// ---- POUs/MAIN.TcPOU
PROGRAM MAIN
VAR
	fbXTSSystem : XTS_System;
	bInit		: BOOL := FALSE;
	i : UDINT;
END_VAR

IF bInit = FALSE THEN
	
		fbXTSSystem.stCfg.bInvertPolarity						:= FALSE;
	
		fbXTSSystem.stCfg.udiNumStations						:= 7;
		fbXTSSystem.stCfg.stStationsCfg[1].sName			 	:= 'Station 1'; 
		fbXTSSystem.stCfg.stStationsCfg[1].lrStartPosition 		:= 0.0; 
		fbXTSSystem.stCfg.stStationsCfg[1].lrEndPosition	 	:= 500.0; 
		fbXTSSystem.stCfg.stStationsCfg[1].lrStopPosition[1] 	:= 100.0; 
		fbXTSSystem.stCfg.stStationsCfg[1].lrStopPosition[2] 	:= 350.0; 
		fbXTSSystem.stCfg.stStationsCfg[1].lrProcessingTime 	:= 2.0;
		fbXTSSystem.stCfg.stStationsCfg[1].uiNumStopPositions 	:= 2;
		fbXTSSystem.stCfg.stStationsCfg[1].lrTravelTime			:= 0.5;				

		fbXTSSystem.stCfg.stStationsCfg[2].sName			 	:= 'Station 2'; 		
		fbXTSSystem.stCfg.stStationsCfg[2].lrStartPosition 		:= 1000.0; 
		fbXTSSystem.stCfg.stStationsCfg[2].lrEndPosition	 	:= 1500.0;
		fbXTSSystem.stCfg.stStationsCfg[2].lrStopPosition[1]	:= 10.0; 
		fbXTSSystem.stCfg.stStationsCfg[2].lrStopPosition[2]	:= 400.0; 
		fbXTSSystem.stCfg.stStationsCfg[2].lrStopPosition[3]	:= 500.0; 
		fbXTSSystem.stCfg.stStationsCfg[2].lrProcessingTime 	:= 3.0;
		fbXTSSystem.stCfg.stStationsCfg[2].uiNumStopPositions 	:= 2;
		fbXTSSystem.stCfg.stStationsCfg[2].lrTravelTime			:= 0.5;				

 		fbXTSSystem.stCfg.stStationsCfg[3].sName			 	:= 'Station 3';  
		fbXTSSystem.stCfg.stStationsCfg[3].lrStartPosition 		:= 2000.0; 
		fbXTSSystem.stCfg.stStationsCfg[3].lrEndPosition	 	:= 2500.0;
		fbXTSSystem.stCfg.stStationsCfg[3].lrStopPosition[1] 	:= 100.0; 
		fbXTSSystem.stCfg.stStationsCfg[3].lrProcessingTime 	:= 1.0;
		fbXTSSystem.stCfg.stStationsCfg[3].uiNumStopPositions 	:= 1;
		fbXTSSystem.stCfg.stStationsCfg[3].lrTravelTime			:= 0.5;				

		fbXTSSystem.stCfg.stStationsCfg[4].sName			 	:= 'Station 4'; 	
		fbXTSSystem.stCfg.stStationsCfg[4].lrStartPosition 		:= 3000.0; 
		fbXTSSystem.stCfg.stStationsCfg[4].lrEndPosition	 	:= 3500.0;
		fbXTSSystem.stCfg.stStationsCfg[4].lrStopPosition[1] 	:= 200.0; 
		fbXTSSystem.stCfg.stStationsCfg[4].lrProcessingTime 	:= 1.0;
		fbXTSSystem.stCfg.stStationsCfg[4].uiNumStopPositions 	:= 1;
		fbXTSSystem.stCfg.stStationsCfg[4].lrTravelTime			:= 0.5;				

		fbXTSSystem.stCfg.stStationsCfg[5].sName			 	:= 'Station 5'; 
		fbXTSSystem.stCfg.stStationsCfg[5].lrStartPosition 		:= 4000.0; 
		fbXTSSystem.stCfg.stStationsCfg[5].lrEndPosition	 	:= 4500.0;
		fbXTSSystem.stCfg.stStationsCfg[5].lrStopPosition[1] 	:= 300.0; 
		fbXTSSystem.stCfg.stStationsCfg[5].lrProcessingTime 	:= 1.0;
		fbXTSSystem.stCfg.stStationsCfg[5].uiNumStopPositions 	:= 1;
		fbXTSSystem.stCfg.stStationsCfg[5].lrTravelTime			:= 0.5;				

		fbXTSSystem.stCfg.stStationsCfg[6].sName			 	:= 'Station 6'; 
		fbXTSSystem.stCfg.stStationsCfg[6].lrStartPosition 		:= 5000.0; 
		fbXTSSystem.stCfg.stStationsCfg[6].lrEndPosition	 	:= 5500.0;
		fbXTSSystem.stCfg.stStationsCfg[6].lrStopPosition[1] 	:= 25.0; 
		fbXTSSystem.stCfg.stStationsCfg[6].lrStopPosition[2] 	:= 325.0; 
		fbXTSSystem.stCfg.stStationsCfg[6].lrStopPosition[3] 	:= 500.0; 
		fbXTSSystem.stCfg.stStationsCfg[6].lrProcessingTime 	:= 3.0;
		fbXTSSystem.stCfg.stStationsCfg[6].uiNumStopPositions 	:= 2;
		fbXTSSystem.stCfg.stStationsCfg[6].lrTravelTime			:= 0.5;				

		fbXTSSystem.stCfg.stStationsCfg[7].sName			 	:= 'Station 7'; 
		fbXTSSystem.stCfg.stStationsCfg[7].lrStartPosition 		:= 6000.0; 
		fbXTSSystem.stCfg.stStationsCfg[7].lrEndPosition	 	:= 6500.0;	
		fbXTSSystem.stCfg.stStationsCfg[7].lrStopPosition[1] 	:= 50.0; 
		fbXTSSystem.stCfg.stStationsCfg[7].lrStopPosition[2] 	:= 450.0;
		fbXTSSystem.stCfg.stStationsCfg[7].lrStopPosition[3] 	:= 500.0;
		fbXTSSystem.stCfg.stStationsCfg[7].lrProcessingTime 	:= 3.0;
		fbXTSSystem.stCfg.stStationsCfg[7].uiNumStopPositions 	:= 2;
		fbXTSSystem.stCfg.stStationsCfg[7].lrTravelTime			:= 0.5;
		
		fbXTSSystem.bEnable := TRUE;

		bInit := TRUE;				
END_IF

XTSSYSTEM();

ACTION XTSSYSTEM:
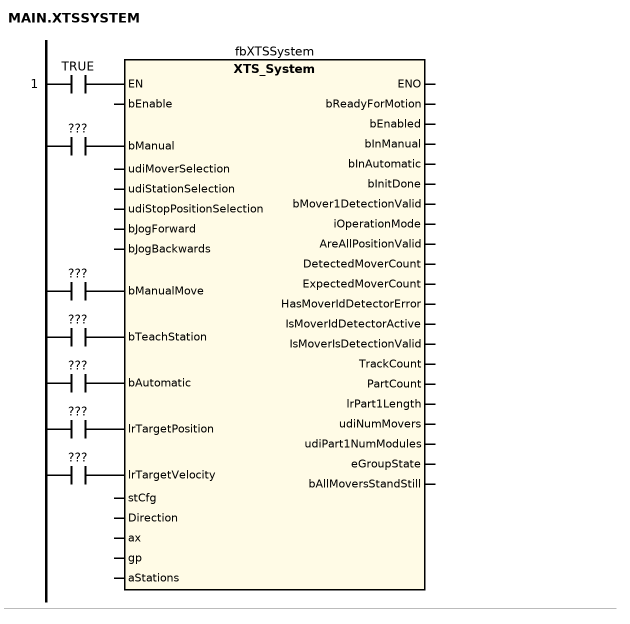
// NETWORK 1
fbXTSSystem(); // XTS_System
END_ACTION

END_PROGRAM

// ---- POUs/XTS/XTS_System.TcPOU
FUNCTION_BLOCK XTS_System
VAR_INPUT
{attribute 'pingroup' := 'Power'}
	bEnable					: BOOL := FALSE;	//Enable operation (power movers, group all ...)
{attribute 'pingroup' := 'Power'}
	bReset					: BOOL := FALSE;	//Reset all axis
{attribute 'pingroup' := 'Manual'}
	bManual					: BOOL;				//Manual operation mode for movers test with collision avoidance
{attribute 'pingroup' := 'Manual'}
	udiMoverSelection		: UDINT := 0;		//Mover ID to move in manual mode. If ID is equal to zero all movers are moved
{attribute 'pingroup' := 'Manual'}
	udiStationSelection		: UDINT := 0;		//Target Station ID for mover selected. If zero manual mode works with target position input
{attribute 'pingroup' := 'Manual'}
	udiStopPositionSelection: UDINT := 1;		//Target Stop Position 1, 2 or 3
{attribute 'pingroup' := 'Manual'}
	bJogForward				: BOOL;				//Jog Forward command for manual mode operation 0
{attribute 'pingroup' := 'Manual'}
	bJogBackwards			: BOOL;				//Jog Backwards command for manual mode operation 0
{attribute 'pingroup' := 'Manual'}
	bManualMove				: BOOL;				//Move selected mover to target position at target velocity in manual mode operation 1
{attribute 'pingroup' := 'Manual'}
	bTeachStation			: BOOL;				//During manual mode flag up of teach station set the stop position of station equal to act mover position
{attribute 'pingroup' := 'Automatic'}
	bAutomatic				: BOOL;				//Automatic operation using stations
{attribute 'pingroup' := 'Profile'}
	lrTargetPosition		: LREAL := 0.0;		//Target Position [mm]
{attribute 'pingroup' := 'Profile'}
	lrTargetVelocity		: LREAL := 500.0;	//Target Velocity [mm]
{attribute 'pingroup' := 'Configuration'}
	stCfg					: stXTSCfg;			//General Configuration
{attribute 'pingroup' := 'Profile'}
	Direction				: tc3_mc3definitions.MC_DIRECTION := tc3_mc3definitions.MC_DIRECTION.mcDirectionPositive;	//Movement Direction	
{attribute 'pingroup' := 'SubElements'}
	ax						: ARRAY [1..Tc3_XTS_Utility.TcIoXtsEnvironmentParameterList.MaxXtsMoversPerXpu] OF FB_Mover;	//Movers
{attribute 'pingroup' := 'SubElements'}
	gp						: FB_GroupCA; //Group CA
{attribute 'pingroup' := 'SubElements'}
	aStations				: ARRAY [1..Tc3_XTS_Utility.TcIoXtsEnvironmentParameterList.MaxXtsInfoStation] OF FB_Station; //Stations
END_VAR
VAR_OUTPUT
{attribute 'pingroup' := 'Status'}
	sLog			 			: STRING := 'Invalid';
{attribute 'pingroup' := 'Status'}
	bError			 			: BOOL;
{attribute 'pingroup' := 'Status'}
	bReadyForMotion 			: BOOL;
{attribute 'pingroup' := 'Status'}
	bEnabled					: BOOL;
{attribute 'pingroup' := 'Manual'}
	bInManual					: BOOL;
{attribute 'pingroup' := 'Automatic'}
	bInAutomatic				: BOOL;
{attribute 'pingroup' := 'XPU'}
	bInitDone					: BOOL;
{attribute 'pingroup' := 'XPU'}
	bMover1DetectionValid 		: BOOL;
{attribute 'pingroup' := 'XPU'}
	iOperationMode 				: OperationMode;
{attribute 'pingroup' := 'XPU'}
	AreAllPositionValid 		: BOOL;
{attribute 'pingroup' := 'XPU'}
	DetectedMoverCount 			: UDINT;
{attribute 'pingroup' := 'XPU'}
	ExpectedMoverCount 			: UDINT;
{attribute 'pingroup' := 'XPU'}
	HasMoverIdDetectorError		: BOOL;
{attribute 'pingroup' := 'XPU'}
	IsMoverIdDetectorActive		: BOOL;
{attribute 'pingroup' := 'XPU'}
	IsMoverIsDetectionValid		: BOOL;
{attribute 'pingroup' := 'XPU'}
	TrackCount					: UDINT;	
{attribute 'pingroup' := 'XPU'}
	PartCount					: UDINT;				
{attribute 'pingroup' := 'XPU'}
	lrPart1Length 				: LREAL;
{attribute 'pingroup' := 'XPU'}
	udiNumMovers  				: UDINT;
{attribute 'pingroup' := 'XPU'}
	udiPart1NumModules			: UDINT;
{attribute 'pingroup' := 'GROUP CA'}
	eGroupState					: MC_GROUP_STATE;
{attribute 'pingroup' := 'GROUP CA'}
	bAllMoversStandStill		: BOOL;	
END_VAR
VAR
	(* XPU *)
	//{attribute 'hide'} 
	fbXTSEnv		 		: FB_TcIoXtsEnvironment;
	//{attribute 'hide'} 
	IXPU			 		: I_TcIoXtsProcessingUnit;
	//{attribute 'hide'} 
	IPart1			 		: I_TcIoXtsXpuPart;
	//{attribute 'hide'} 
	fbInfoServer			: FB_TcIoXtsInfoServer;
	//{attribute 'hide'} 
	aInfoServerOids			: ARRAY [1..Tc3_XTS_Utility.TcIoXtsEnvironmentParameterList.MaxXtsInfoServer] OF Tc3_XTS_Utility.OTCID;
	//{attribute 'hide'} 
	aStationsOTCID			: ARRAY [1..Tc3_XTS_Utility.TcIoXtsEnvironmentParameterList.MaxXtsInfoStation] OF Tc3_XTS_Utility.OTCID;
	//{attribute 'hide'} 
	aMoversOids				: ARRAY [1..Tc3_XTS_Utility.TcIoXtsEnvironmentParameterList.MaxXtsMoversPerXpu] OF Tc3_XTS_Utility.OTCID;
	//{attribute 'hide'} 
	GroupCAOTCID			: ARRAY [1..Tc3_XTS_Utility.TcIoXtsEnvironmentParameterList.MaxXtsCaGroup] OF Tc3_XTS_Utility.OTCID;
END_VAR
VAR
	bXPUInitDone			: BOOL;
	stVisuStationsCfg 		: ARRAY [1..Tc3_XTS_Utility.TcIoXtsEnvironmentParameterList.MaxXtsInfoStation] OF stStationCfg;
END_VAR


//Initialization
Init(); 

//Operation
IF bInitDone THEN
	//Enable System
	bEnabled := Enable(bEnable);
	bInManual:= Manual(bManual AND bInAutomatic = FALSE AND bEnabled);
	bInAutomatic := Automatic(bAutomatic AND bInManual = FALSE AND bEnabled);
	gp.m_reset(bReset);
	//bConfigurationDone := Configuration(bApplyConfiguration);
END_IF
IF udiNumMovers <> 0 THEN
	//Call sub fb's like group CA, movers...
	Childs();
	//Status
	bReadyForMotion := gp.bError = FALSE AND bEnabled;
	bError			:= gp.bError;
END_IF

METHOD PRIVATE Automatic : BOOL
VAR_INPUT
	bEnable : BOOL;
END_VAR
VAR_INST
	iState 		: INT;
	bAllDone 	: BOOL;
	i 			: UDINT;
	bBusy		: BOOL;
END_VAR

CASE iState OF
	
	0 : IF bEnable THEN 
			iState := iState + 1; 
			bBusy  := TRUE;
		END_IF
		
	1 : //Move all to zero position
		bAllDOne := FALSE;
		FOR i:= 1 TO udiNumMovers DO
			bAllDone := bAllDOne OR ax[i].m_moveca(TRUE, 0.0, 1000.0);
		END_FOR
		IF bAllMoversStandStill AND bAllDone THEN
			FOR i:= 1 TO udiNumMovers DO
				ax[i].m_moveca(FALSE, 0.0, 0.0);
			END_FOR
			iState := iState + 1;
		END_IF
		IF bEnable = FALSE THEN iState := iState + 1; END_IF
	
	2 : //Start
		bAllDOne := TRUE;
		FOR i:= 1 TO udiNumMovers DO
			bAllDone := bAllDOne AND ax[i].Sequence1(TRUE);
		END_FOR
		IF bEnable = FALSE THEN iState := iState + 1; END_IF
	
	3 : //Stop
		bAllDOne := TRUE;
		FOR i:= 1 TO udiNumMovers DO
			bAllDone := bAllDOne AND NOT ax[i].Sequence1(FALSE);
		END_FOR
		IF bAllDone THEN
			iState := iState + 1;
		END_IF
		
	4 : bBusy := FALSE;
		IF bEnable = FALSE THEN
			iState := 0;
		END_IF
		
END_CASE
Automatic := bBusy;
END_METHOD

METHOD PRIVATE Childs : BOOL
VAR_INPUT
END_VAR
VAR_INST
	i 	: UDINT;
	bAllDone : BOOL;
END_VAR
//Call Group CA
gp(ax:= ax, eGroupState=> eGroupState, bAllStandStill=> bAllMoversStandStill, bError=> );
//Call Movers
FOR i := 1 TO udiNumMovers DO
	ax[i](aStations := aStations, udiID=> );
END_FOR
//Call Stations
FOR i:= 1 TO stCfg.udiNumStations DO
	aStations[i]();
END_FOR
END_METHOD

METHOD Configuration : BOOL
VAR_INPUT
	bExecute : BOOL;
END_VAR
VAR_INST
	i : UDINT;
	bDone : BOOL;
END_VAR
FOR i:= 1 TO stCfg.udiNumStations DO
	bDone := bExecute;
	bDone := bDone AND aStations[i].SetStationInfo(bExecute, OTCID := aStationsOTCID[i]);
END_FOR
Configuration := bDone;
END_METHOD

METHOD PRIVATE Enable : BOOL
VAR_INPUT
	bEnable		: BOOL;
END_VAR
VAR_INST
	iState 		: INT;
	bAllDone 	: BOOL;
	i 			: UDINT;
	bDone		: BOOL;
END_VAR

CASE iState OF
	
	0 : 
		IF bEnable THEN 
			FOR i := 1 TO udiNumMovers DO
				ax[i].m_ClearCmd();
			END_FOR
			gp.m_clearcmd();
			bDone := FALSE;
			iState := iState + 10; 
		END_IF
	
	10 : //
		bAllDone := TRUE;
		FOR i := 1 TO udiNumMovers DO
			bAllDone := bAllDone AND ax[i].m_reset(TRUE);
		END_FOR
		IF bAllDone THEN
			iState := iState + 10;
		END_IF
		
	20 : //Power all Axis
		bAllDone := TRUE;
		FOR i := 1 TO udiNumMovers DO
			bAllDone := bAllDone AND ax[i].m_power_on();
		END_FOR
		IF bAllDone THEN
			iState := iState + 10;
		END_IF
		
	30 : //Reset Group
		IF gp.m_reset(TRUE) THEN
			iState := iState + 10;
		END_IF
		
	40 : //Add all axis to group
		bAllDone := TRUE;
		FOR i := 1 TO udiNumMovers DO
			bAllDone := bAllDone AND ax[i].m_add2Group(TRUE, ag := gp.ag);
		END_FOR
		IF bAllDone THEN
			FOR i := 1 TO udiNumMovers DO
				ax[i].m_add2Group(FALSE, ag := gp.ag);
			END_FOR
			iState := iState + 10;
		END_IF
		
	50 : //Enable group
		IF gp.m_enable(TRUE) THEN
			iState := iState + 10;
		END_IF
		
	60 : //Jog Done
		 bDone := TRUE;
		 IF bEnable = FALSE THEN iState := 70; END_IF 

	70 : //Halt group
		bAllDone := TRUE;
		FOR i := 1 TO udiNumMovers DO
			bAllDone := bAllDone AND ax[i].m_haltca(TRUE);
		END_FOR
		IF bAllDone THEN
			iState := iState + 10;
		END_IF
		
	80 : //Disable
		IF gp.m_disable(TRUE) THEN
			iState := iState + 10;
		END_IF		

	90 : //UnGroup
		IF gp.m_ungroupall(TRUE) THEN
			iState := iState + 10;
		END_IF
	
	100 : //Power off all
		bAllDone := TRUE;
		FOR i := 1 TO udiNumMovers DO
			bAllDone := bAllDone AND ax[i].m_power_off();
		END_FOR
		IF bAllDone THEN
			bDone := FALSE;
			iState := 0;
		END_IF
		 
END_CASE
Enable := bDone;
END_METHOD

METHOD PRIVATE Init
VAR_INST
	iState 		: INT;
	bAllDone 	: BOOL;
	i 			: UDINT;
END_VAR

//XPU Initialization
IF bXPUInitDone = FALSE THEN
	sLog := 'Init: Initialazing XPU';
	IF fbXTSEnv.Init(TRUE) THEN
		sLog := 'Init: XPU Initialazed';
		fbXTSEnv.Init(FALSE);
		bXPUInitDone := TRUE;
	END_IF	
END_IF

CASE iState OF
	
	0 : 
		IF bXPUInitDone THEN iState := iState + 10; END_IF
	
	10 : //Get XPU Parameters
		sLog := 'Init: Checking XPU parameters';
		Ixpu 						:= fbXTSEnv.XpuTcIo(1);
		IPart1						:= Ixpu.PartTcIo(1);
		iOperationMode 				:= Ixpu.GetOperationMode();
		AreAllPositionValid 		:= Ixpu.GetAreAllPositionsValid();
		DetectedMoverCount 			:= Ixpu.GetDetectedMoverCount();
		ExpectedMoverCount 			:= Ixpu.GetExpectedMoverCount();
		HasMoverIDDetectorError 	:= Ixpu.GetHasMoverIdDetectionError();
		IsMoveriddetectoractive 	:= Ixpu.GetIsMoverIdDetectionActive();
		ismoverisdetectionvalid 	:= Ixpu.GetIsMoverIdDetectionValid();
		TrackCount					:= Ixpu.GetTrackCount();
		PartCount					:= Ixpu.GetPartCount();
		lrPart1Length 				:= IPart1.GetLength();
		udiPart1NumModules			:= IPart1.GetModuleCount();
		udiNumMovers 				:= Ixpu.GetMoverCount();
		
		IF (Ixpu.GetDetectedMoverCount() = Ixpu.GetExpectedMoverCount()) AND Ixpu.GetAreAllPositionsValid() THEN
			iState := iState + 10; 			
		END_IF

	20 : //Detect Mover 1 
		sLog := 'Init: Detecting mover 1';
		IF Ixpu.GetIsMoverIdDetectionValid() = FALSE THEN
			IF Ixpu.GetMoverIdDetectionMode() = 1 THEN
				Ixpu.TriggerMoverIdDetection();
				iState := iState + 1;
			ELSE
				bMover1DetectionValid := TRUE;
				iState := iState + 10;
			END_IF
		ELSE
			bMover1DetectionValid := TRUE;
			iState := iState + 10;
		END_IF
		
	21 : //Check Mover 1 Detection Valid
		IF Ixpu.GetIsMoverIdDetectionValid() THEN
			bMover1DetectionValid := TRUE;
			iState := 30;
		END_IF
	
	30 : //Get OIDS of Group CA
		sLog := 'Init: Getting group CA Oids';
		IF fbXTSEnv.GetCaGroupOids(TRUE) THEN
			fbXTSEnv.GetCaGroupOids(FALSE);
			GroupCAOTCID := fbXTSEnv.P_CaGroupOids;
			gp.fbXPUGroupCA.Init(FALSE, GroupCAOTCID[1]);
			iState := 31;
		END_IF
		
	31 : //Reset Group
		sLog := 'Init: Resseting group CA';
		IF gp.m_reset(TRUE) THEN
			gp.m_reset(FALSE);
			iState := iState + 1;
		END_IF
		
	32 : //Disable Group in order to configure the Rail Length
		sLog := 'Init: UnGroup all';
		IF gp.m_ungroupall(TRUE) THEN
			gp.m_ungroupall(FALSE);
			iState := iState + 1;
		END_IF
		
	33 : //Set Group CA Rail Length equal to Part 1 length
		sLog := 'Init: Get group CA Oids';
		IF gp.fbXPUGroupCA.Init(TRUE, GroupCAOTCID[1]) THEN
			IF gp.fbXPUGroupCA.SetRailLength(lrPart1Length) THEN
				gp.fbXPUGroupCA.Init(FALSE, GroupCAOTCID[1]);
				iState := 40;		
			END_IF
		END_IF
		
	40 : //Get Info Server OIDS
		sLog := 'Init: Get Info Server Oids';
		IF Tc3_XTS_Utility.TcIoXtsEnvironmentParameterList.MaxXtsInfoServer > 0 THEN 
			IF fbXTSEnv.GetInfoServerOids(TRUE) THEN
				fbXTSEnv.GetInfoServerOids(FALSE);
				aInfoServerOids := fbXTSEnv.P_InfoServerOids;
				i:=1;
				fbInfoServer.Init(FALSE, aInfoServerOids[i]);
				iState := iState + 1;
			END_IF
		ELSE
			iState := iState + 10;
		END_IF

	41 : //Get OCID of Stations
		sLog := 'Init: Get Info Stations Oids';
		IF fbInfoServer.Init(TRUE, aInfoServerOids[i]) THEN
			IF fbInfoServer.GetInfoStationOids() THEN
				aStationsOTCID := fbInfoServer.P_InfoStationOids;
				fbInfoServer.Init(FALSE, aInfoServerOids[i]);
				FOR i:= 1 TO stCfg.udiNumStations DO
					aStations[i].SetStationInfo(FALSE, OTCID := aStationsOTCID[i]);
				END_FOR
				iState := 50;
			END_IF
		END_IF
		
	50 : //Get Mover OIDS
		sLog := 'Init: Get movers Oids';
		IF IXPU.GetMoverOids() THEN
			aMoversOids := IXPU.P_MoverOids;
			iState := iState + 1;
		END_IF
		
	51 : //Reset Movers
		sLog := 'Init: Reset movers';
		bAllDOne := TRUE;
		 FOR i := 1 TO udiNumMovers DO
			 bAllDone := bAllDone AND ax[i].m_reset(TRUE);
		 END_FOR
		 IF bAllDOne THEN
			 FOR i := 1 TO udiNumMovers DO
			 	ax[i].m_reset(FALSE);
		 	 END_FOR
			 iState := iState + 1;
		 END_IF
		 
	52 : //Power off Movers
		sLog := 'Init: Power off movers';
		bAllDOne := TRUE;
		 FOR i := 1 TO udiNumMovers DO
			 bAllDone := bAllDone AND ax[i].m_power_off();
		 END_FOR
		 IF bAllDOne THEN
			 iState := iState + 1;
		 END_IF
		 
	53 : //Configure Movers
		sLog := 'Init: Configure movers';
		 bAllDone := TRUE;
		 FOR i := 1 TO udiNumMovers DO
			 bAllDone := bAllDone AND ax[i].m_InvertPolarity(TRUE, stCfg.bInvertPolarity);
		 END_FOR
	 	IF bAllDOne THEN
			 FOR i := 1 TO udiNumMovers DO
			 	ax[i].m_InvertPolarity(FALSE, stCfg.bInvertPolarity);
		 	 END_FOR
			 iState := 60;
	 	END_IF
		
	60 : //Set Stations configuration
		sLog := 'Init: Configure stations';
		bAllDone := TRUE;
		FOR i:= 1 TO stCfg.udiNumStations DO
			aStations[i](stCfg := stCfg.stStationsCfg[i], (*ax := ax,*) udiNumMovers := udiNumMovers, lrPartLength := lrPart1Length, bInvertPolarity := stCfg.bInvertPolarity);
			IF Tc3_XTS_Utility.TcIoXtsEnvironmentParameterList.MaxXtsInfoStation > 0 AND Tc3_XTS_Utility.TcIoXtsEnvironmentParameterList.MaxXtsInfoServer > 0 THEN 
				bAllDone := bAllDone AND aStations[i].SetStationInfo(TRUE, OTCID := aStationsOTCID[i]);
			ELSE
				bAllDone := TRUE;
			END_IF
			(*IF i<stCfg.udiNumStations THEN
				aStations[i].lrNextPosition := stCfg.stStationsCfg[i+1].lrStartPosition;	
			ELSIF i = stCfg.udiNumStations THEN	
				aStations[i].lrNextPosition := stCfg.stStationsCfg[1].lrStartPosition;	
			END_IF
			IF i=1 THEN
				aStations[i].lrPreviousEndPosition := stCfg.stStationsCfg[stCfg.udiNumStations].lrEndPosition;	
			ELSE
				aStations[i].lrPreviousEndPosition := stCfg.stStationsCfg[i-1].lrEndPosition;	
			END_IF*)
			IF bAllDone THEN
				iState := 70;
			END_IF
		END_FOR
		
	70 : //Jog Done
		 sLog := 'Init: Done!';
		 bInitDone 	:= TRUE;
			 
END_CASE
END_METHOD

METHOD PRIVATE Manual : BOOL
VAR_INPUT
	bEnable 			: BOOL;
END_VAR
VAR_INST
	iState 				: INT;
	bAllDone 			: BOOL;
	i 					: UDINT;
	bBusy				: BOOL;
	fbRTRIG				: R_Trig;
END_VAR

CASE iState OF
	0 : IF bEnable THEN 
			iState := iState + 1; 
			bBusy  := TRUE;
		END_IF
		
	1 : //Idle
		IF bEnable = FALSE THEN
			iState := 100;
		ELSIF bJogBackwards OR bJogForward THEN
			iState := 10; 
		ELSIF bManualMove AND udiStationSelection = 0 THEN
			//Move All with Target Position
			iState := 50; 
		ELSIF bManualMove AND udiStationSelection > 0 AND udiStationSelection < stCfg.udiNumStations+1 AND udiStopPositionSelection > 0 AND udiStopPositionSelection < 4 THEN
			//Move Mover to Station 
			iState := 60;
		ELSIF bTeachStation AND udiStationSelection > 0 AND udiMoverSelection > 0 AND udiStopPositionSelection > 0 AND udiStopPositionSelection < 4 THEN
			iState := 70;
		END_IF
		
	10 : //Manual mode operation 0 
		IF udiMoverSelection = 0 THEN
			bAllDone := TRUE;
			FOR i := 1 TO udiNumMovers DO
				bAllDone := bAllDone AND ax[i].m_jogca_velo(bJogBackwards, bJogForward, lrTargetVelocity) = FALSE;
			END_FOR
			IF bJogBackwards = FALSE AND bJogForward = FALSE AND bAllDone THEN
				iState := 1;
			END_IF	
		ELSE
			IF udiMoverSelection < 1 OR udiMoverSelection > udiNumMovers THEN udiMoverSelection := 1; END_IF
			IF ax[udiMoverSelection].m_jogca_velo(bJogBackwards, bJogForward, lrTargetVelocity) = FALSE AND bJogBackwards = FALSE AND bJogForward = FALSE THEN
				iState := 1;	
			END_IF
		END_IF
		
	50 : //Manual Operation with Target Position
		IF udiMoverSelection = 0 THEN
			FOR i := 1 TO udiNumMovers DO
				ax[i].m_moveca_direction(bManualMove, lrTargetPosition, lrTargetVelocity, Direction);
			END_FOR
			IF bAllMoversStandStill AND bManualMove = FALSE THEN
				iState := 1;
			END_IF
		ELSE ax[udiMoverSelection].m_moveca_direction(bManualMove, lrTargetPosition, lrTargetVelocity, Direction);
			IF bAllMoversStandStill AND bManualMove = FALSE THEN
				iState := 1;
			END_IF
		END_IF
		
	60 : //Manual Operation with Stations
		IF udiMoverSelection = 0 THEN
			FOR i := 1 TO udiNumMovers DO
				ax[i].m_moveca_direction(bManualMove, aStations[udiStationSelection].stCfg.lrStopPosition[udiStopPositionSelection] + aStations[udiStationSelection].stCfg.lrStartPosition, lrTargetVelocity, Direction);
			END_FOR
			IF bAllMoversStandStill AND bManualMove = FALSE THEN
				iState := 1;
			END_IF
		ELSE ax[udiMoverSelection].m_moveca_direction(bManualMove, aStations[udiStationSelection].stCfg.lrStopPosition[udiStopPositionSelection] + aStations[udiStationSelection].stCfg.lrStartPosition, lrTargetVelocity, Direction);
			IF bAllMoversStandStill AND bManualMove = FALSE THEN
				iState := 1;
			END_IF
		END_IF
		
	70 : //Teach Station
		stCfg.stStationsCfg[udiStationSelection].lrStopPosition[udiStopPositionSelection] := ax[udiMoverSelection].p_Axis.NcToPlc.ModuloSetPos-stCfg.stStationsCfg[udiStationSelection].lrStartPosition;
		bAllDone := TRUE;	
		FOR i:= 1 TO stCfg.udiNumStations DO
			bAllDone := bAllDone AND aStations[i].SetStationInfo(TRUE, OTCID := aStationsOTCID[i]);
		END_FOR
		IF bAllDone THEN
			FOR i:= 1 TO stCfg.udiNumStations DO
				aStations[i].SetStationInfo(FALSE, OTCID := aStationsOTCID[i]);
			END_FOR
			iState := iState + 1;
		END_IF
		
	71 : //Apply New Configuration
		IF bTeachStation = FALSE THEN
			iState := 1;
		END_IF
		
	100 : 
		bBusy := FALSE;
		iState := 0;
		
END_CASE
Manual := bBusy;
END_METHOD

END_FUNCTION_BLOCK

// ---- POUs/XTS/FB_Mover.TcPOU
FUNCTION_BLOCK FB_Mover 
VAR_IN_OUT
	aStations				: ARRAY [1..Tc3_XTS_Utility.TcIoXtsEnvironmentParameterList.MaxXtsInfoStation] OF FB_Station; //Stations
END_VAR
VAR_OUTPUT
	udiID					: UDINT;
END_VAR
VAR
	//Function Blocks
	fbCtcIoXTSMover			: FB_TcIoXtsXPUMover;
	ax						: AXIS_REF;
	fbPower 				: MC_Power;
	fbReset 				: MC_Reset;
	fbHaltCA				: MC_HaltCA;
	fbMoveAbsCA				: MC_MoveAbsoluteCA;
	fbMoveRelCA				: MC_MoveRelativeCA;
	fbMoveAbsTimeCA			: MC_MoveAbsoluteTimeCA;
	fbMoveAbs				: MC_MoveAbsolute;
	fbGearIn				: MC_GearIn;
	fbGearOut				: MC_GearOut;
	fbReadParamSet			: MC_ReadParameterSet := (Execute := TRUE);
	fbAddAxis2Group 		: MC_AddAxisToGroup;
	stParameter				: ST_AxisParameterSet;
	fbJogCA					: MC_JOGCA;
	fbJog					: MC_Jog;
END_VAR

ax.ReadStatus();

fbPower(
	Axis:= ax, 
	Enable:= , 
	Enable_Positive:= , 
	Enable_Negative:= , 
	Override:= , 
	BufferMode:= , 
	Options:= , 
	Status=> , 
	Busy=> , 
	Active=> , 
	Error=> , 
	ErrorID=> );
	
fbReset(
	Axis:= ax, 
	Execute:= , 
	Busy=> , 
	Done=> ,
	Error=> , 
	ErrorID=> );
	
fbJog(
	Axis:= ax, 
	JogForward:= , 
	JogBackwards:= , 
	Mode:= , 
	Position:= , 
	Velocity:= , 
	Acceleration:= , 
	Deceleration:= , 
	Jerk:= , 
	Done=> , 
	Busy=> , 
	Active=> , 
	CommandAborted=> , 
	Error=> , 
	ErrorID=> );

fbJogCA(
	Axis:= ax, 
	JogForward:= , 
	JogBackwards:= , 
	Mode:= , 
	Position:= , 
	Velocity:= , 
	Acceleration:= , 
	Deceleration:= , 
	Jerk:= , 
	Done=> , 
	Busy=> , 
	Active=> , 
	CommandAborted=> , 
	Error=> , 
	ErrorID=> );
	
fbMoveAbsCA(
	Axis:= ax, 
	Execute:= , 
	ContinuousUpdate:= , 
	Position:= , 
	Velocity:= , 
	Acceleration:= , 
	Deceleration:= , 
	Jerk:= , 
	Gap:= , 
	BufferMode:= , 
	Direction:= , 
	Options:= , 
	Busy=> , 
	Done=> ,
	Error=> , 
	ErrorID=> );
	
fbMoveAbsTimeCA(
	Axis:= ax, 
	bExecute:= , 
	lrPosition:= , 
	lrTime:= , 
	Done=> , 
	Busy=> , 
	Active=> , 
	CommandAborted=> , 
	Error=> , 
	ErrorId=> );
	
fbHaltCA(
	Axis:= ax, 
	Execute:= , 
	Deceleration:= , 
	Jerk:= , 
	Options:= , 
	Busy=> , 
	Done=> ,
	Error=> , 
	ErrorID=> );

fbMoveAbs(
	Axis:= ax, 
	Execute:= , 
	Position:= , 
	Velocity:= , 
	Acceleration:= , 
	Deceleration:= , 
	Jerk:= , 
	BufferMode:= , 
	Options:= , 
	Busy=> , 
	Done=> ,
	Error=> , 
	ErrorID=> );
	
fbMoveRelCA(
	Axis:= ax, 
	Execute:= , 
	ContinuousUpdate:= , 
	Distance:= , 
	Velocity:= , 
	Acceleration:= , 
	Deceleration:= , 
	Jerk:= , 
	Gap:= , 
	BufferMode:= , 
	Options:= , 
	Busy=> , 
	Done=> ,
	Error=> , 
	ErrorID=> );
	
fbGearOut(
	Slave:= ax, 
	Execute:= , 
	Options:= , 
	Done=> , 
	Busy=> , 
	Error=> , 
	ErrorID=> );

fbReadParamSet(Parameter := stParameter, Axis := ax);
udiID := stParameter.AxisId;

METHOD m_add2Group : BOOL
VAR_INPUT
	bExecute	: BOOL;
	ag		 	: AXES_GROUP_REF;
END_VAR
fbAddAxis2Group(
	AxesGroup:= ag, 
	Axis:= ax, 
	Execute:= bExecute, 
	IdentInGroup:= UDINT_TO_IDENTINGROUP(ax.NcToPlc.AxisId), 
	Done=> m_Add2Group, 
	Busy=> , 
	Error=> , 
	ErrorId=> );
END_METHOD

METHOD m_clearCmd : BOOL
VAR_INPUT
END_VAR
fbMoveAbsCA.Execute := FALSE;
fbHaltCA.Execute := FALSE;
fbGearIn.Execute := FALSE;
fbReset.Execute	:= FALSE;
END_METHOD

METHOD m_gearIn : BOOL
VAR_INPUT
	bExecute 			: BOOL;
	lrRatioNumerator 	: LREAL;
	uiRatioDenominator	: UINT;
END_VAR
VAR_IN_OUT
	axMaster	: AXIS_REF;	
END_VAR
fbGearIn.Execute 	:= bExecute;
m_gearIn 			:= fbGearIn.InGear;

fbGearIn(
	Master:= axMaster, 
	Slave:= ax, 
	Execute:= , 
	RatioNumerator:= lrRatioNumerator, 
	RatioDenominator:= uiRatioDenominator, 
	Acceleration:= , 
	Deceleration:= , 
	Jerk:= , 
	BufferMode:= , 
	Options:= , 
	InGear=> , 
	Busy=> , 
	Active=> , 
	CommandAborted=> , 
	Error=> , 
	ErrorID=> );
END_METHOD

METHOD m_gearOut : BOOL
VAR_INPUT
	bExecute 			: BOOL;
END_VAR
fbGearOut.Execute 	:= bExecute;
m_gearOut 			:= fbGearOut.Done;
END_METHOD

METHOD m_getmoveratpos : BOOL
VAR_INPUT
	lrPosition : LREAL;
END_VAR
IF ax.NcToPlc.ModuloSetPos > lrPosition-1 AND ax.NcToPlc.ModuloSetPos < lrPosition+1 THEN
	m_getmoveratpos := TRUE;
END_IF
END_METHOD

METHOD m_haltca : BOOL
VAR_INPUT
	bExecute : BOOL;
END_VAR
fbHaltCA.Execute 	:= bExecute;
fbHaltCA.Gap		:= MC_DEFAULT;
m_haltca			:= fbHaltCA.Done;
END_METHOD

METHOD m_InvertPolarity : BOOL
VAR_INPUT
	bExecute : BOOL;
	bValue	 : BOOL;
END_VAR
VAR_INST
	iState 		: INT;
	fbWrite 	: MC_WriteParameterPersistent;
END_VAR

CASE iState OF 
	0 : IF bExecute THEN 
			fbWrite(Axis := ax, Execute := FALSE);
			iState := iState + 1; 
		END_IF
	1 :  
		fbWrite(
			Axis:= ax, 
			Execute:= TRUE, 
			ParameterNumber:= MC_AxisParameter.AxisMotorDirectionInverse, 
			Value:= BOOL_TO_LREAL(bValue), 
			Done=> , 
			Busy=> , 
			Error=> , 
			ErrorID=> );
		IF fbWrite.Done THEN
			fbWrite(Axis := ax, Execute := FALSE);
			iState := iState + 1;
		END_IF
	2 : 
		fbWrite(
			Axis:= ax, 
			Execute:= TRUE, 
			ParameterNumber:= MC_AxisParameter.AxisEncoderDirectionInverse, 
			Value:= BOOL_TO_LREAL(bValue), 
			Done=> , 
			Busy=> , 
			Error=> , 
			ErrorID=> );
		IF fbWrite.Done THEN
			fbWrite(Axis := ax, Execute := FALSE);
			iState := iState + 1;
		END_IF
	3 : //Job Done
		m_InvertPolarity := TRUE;
		IF bExecute = FALSE THEN
			iState := 0;
		END_IF
END_CASE
END_METHOD

METHOD m_jogca : BOOL
VAR_INPUT
	bJogBackwards	: BOOL;
	bJogForward		: BOOL;
END_VAR
fbJogCA.JogBackwards	:= bJogBackwards;
fbJogCA.JogForward		:= bJogForward;
//fbJogCA.Mode		:= eType;
//fbJogCA.Position	:= lrPosition;
//fbJogCA.Velocity	:= lrVelocity;
m_jogca				:= fbJogCA.Busy;
END_METHOD

METHOD m_jogca_velo : BOOL
VAR_INPUT
	bJogBackwards	: BOOL;
	bJogForward		: BOOL;
	lrVelocity		: LREAL;
END_VAR
fbJogCA.JogBackwards	:= bJogBackwards;
fbJogCA.JogForward		:= bJogForward;
fbJogCA.Mode			:= E_JogMode.MC_JOGMODE_CONTINOUS;
fbJogCA.Velocity		:= lrVelocity;
m_jogca_velo			:= fbJogCA.Busy;
END_METHOD

METHOD m_moveca : BOOL
VAR_INPUT
	bExecute	: BOOL;
	lrPosition 	: LREAL;
	lrVelocity	: LREAL;
END_VAR
fbMoveAbsCA.Position 			:= lrPosition;
fbMoveAbsCA.Velocity			:= lrVelocity;
fbMoveAbsCA.Acceleration		:= stParameter.fAcceleration; 
fbMoveAbsCA.Deceleration		:= stParameter.fDeceleration; 
fbMoveAbsCA.Jerk				:= stParameter.fJerk; 
fbMoveAbsCA.Direction			:= tc3_mc3definitions.mcDirectionPositive;
fbMoveAbsCA.ContinuousUpdate 	:= TRUE;
fbMoveAbsCA.Execute				:= bExecute;
fbMoveAbsCA.Gap					:= MC_DEFAULT;
m_moveca						:= fbMoveAbsCA.Done;
END_METHOD

METHOD m_moveca_bytime : BOOL
VAR_INPUT
	bExecute	: bool;
	lrPosition 	: LREAL;
	lrTime		: LREAL;
END_VAR
(*VAR_INST
	fbProfileByTime : FB_ProfileByTime;
END_VAR*)
(*fbProfileByTime.lrDistance := lrPosition - ax.NcToPlc.ModuloSetPos;
IF fbProfileByTime.lrDistance <> 0 THEN
	IF fbProfileByTime.lrDistance < 0 THEN fbProfileByTime.lrDistance := fbProfileByTime.lrDistance + stParameter.fEncModuloFactor; END_IF
	fbProfileByTime(
		lrTime:= lrTime, 
		//lrDistance:= lrPosition - fbAxis.NcToPlc.ModuloSetPos, 
		lrMaxVelocity:= stParameter.fVeloMaximum, 
		lrMaxAcceleration:= stParameter.fAcceleration, 
		lrMaxJerk:= stParameter.fJerk, 
		lrVelocity=> , 
		lrAcceleration=> , 
		lrJerk=> );
		
	fbMoveAbsCA.Position		:= lrPosition;
	fbMoveAbsCA.Direction		:= tc3_mc3Definitions.MC_DIRECTION.mcDirectionPositive;
	fbMoveAbsCA.Velocity 		:= MAX(fbProfileByTime.lrVelocity, 100.0);
	fbMoveAbsCA.Acceleration 	:= fbProfileByTime.lrMaxAcceleration;
	fbMoveAbsCA.Deceleration 	:= fbProfileByTime.lrMaxAcceleration;
	fbMoveAbsCA.Jerk 			:= fbProfileByTime.lrMaxJerk;
	fbMoveAbsCA.Execute			:= bExecute;
	
	IF fbMoveAbsCA.Done THEN
		m_moveca_bytime := TRUE;
	END_IF
ELSE
	m_moveca_bytime := TRUE;
END_IF*)

fbMoveAbsTimeCA.bExecute 	:= bExecute;
fbMoveAbsTimeCA.lrPosition 	:= lrPosition;
fbMoveAbsTimeCA.lrTime		:= lrTime;
m_moveca_bytime				:= fbMoveAbsTimeCA.Done;
END_METHOD

METHOD m_moveca_direction : BOOL
VAR_INPUT
	bExecute	: BOOL;
	lrPosition 	: LREAL;
	lrVelocity	: LREAL;
	Direction	: tc3_mc3definitions.MC_DIRECTION;
END_VAR
fbMoveAbsCA.Position 			:= lrPosition;
fbMoveAbsCA.Velocity			:= lrVelocity;
fbMoveAbsCA.Acceleration		:= stParameter.fAcceleration; 
fbMoveAbsCA.Deceleration		:= stParameter.fDeceleration; 
fbMoveAbsCA.Jerk				:= stParameter.fJerk; 
fbMoveAbsCA.Direction			:= Direction;
fbMoveAbsCA.ContinuousUpdate 	:= TRUE;
fbMoveAbsCA.Execute				:= bExecute;
fbMoveAbsCA.Gap					:= MC_DEFAULT;
m_moveca_direction				:= fbMoveAbsCA.Done;
END_METHOD

METHOD m_moveca_gap : BOOL
VAR_INPUT
	bExecute	: BOOL;
	lrPosition 	: LREAL;
	lrVelocity	: LREAL;
	lrGap		: LREAL;
END_VAR
fbMoveAbsCA.Position 			:= lrPosition;
fbMoveAbsCA.Velocity			:= lrVelocity;
fbMoveAbsCA.Acceleration		:= stParameter.fAcceleration; 
fbMoveAbsCA.Deceleration		:= stParameter.fDeceleration; 
fbMoveAbsCA.Jerk				:= stParameter.fJerk; 
fbMoveAbsCA.Direction			:= tc3_mc3definitions.mcDirectionPositive;
fbMoveAbsCA.ContinuousUpdate 	:= TRUE;
fbMoveAbsCA.Execute				:= bExecute;
fbMoveAbsCA.Gap					:= lrGap;
m_moveca_gap					:= fbMoveAbsCA.Done;
END_METHOD

METHOD m_moverstandstill : BOOL
VAR_INPUT
END_VAR
m_moverstandstill := ax.NcToPlc.SetVelo=0.0;
END_METHOD

METHOD m_power_off : BOOL
VAR_INPUT
END_VAR
fbPower.Enable 			:= FALSE;
fbPower.Enable_Positive := FALSE;
fbPower.Enable_Negative := FALSE;
m_power_off := NOT fbPower.Status;
END_METHOD

METHOD m_power_on : BOOL
fbPower.Enable 			:= TRUE;
fbPower.Enable_Positive := TRUE;
fbPower.Enable_Negative := TRUE;
m_power_on				:= fbPower.Status;
END_METHOD

METHOD m_reset : BOOL
VAR_INPUT
	bExecute : BOOL;
END_VAR
fbReset.Execute			:= bExecute;
m_reset					:= fbReset.Done;
END_METHOD

METHOD m_standstill : BOOL
VAR_INPUT
END_VAR
m_standstill := ax.NcToPlc.SetVelo=0;
END_METHOD

PROPERTY p_Axis : reference to AXIS_REF
GET
p_Axis ref= ax;
END_GET
SET
ax := p_Axis;
END_SET
END_PROPERTY

{warning 'add property implementation'}
PROPERTY p_ModulePos : lreal
GET
p_ModulePos := ax.NcToPlc.ModuloActPos;
END_GET
END_PROPERTY

METHOD Sequence1 : BOOL
VAR_INPUT
	bEnable 	: BOOL;
END_VAR
VAR_INST
	iState 		: INT;
	iStation 	: INT;
	oTON		: TON;
	bBusy		: BOOL;
END_VAR

CASE iState OF

	0 : //Idle
		bBusy := FALSE;
		IF bEnable THEN
			iState := iState + 10;
			bBusy := TRUE;
			iStation := 1;
			m_moveca_bytime(FALSE, 0.0, 0.0);
		END_IF

	10 : //
		 IF m_moveca_bytime(TRUE, aStations[iStation].stCfg.lrStartPosition + aStations[iStation].stCfg.lrStopPosition[1], aStations[iStation].stCfg.lrTravelTime) THEN
			 m_moveca_bytime(FALSE, aStations[iStation].stCfg.lrStartPosition + aStations[iStation].stCfg.lrStopPosition[1], aStations[iStation].stCfg.lrTravelTime);
			 iState := iState + 10;
		 END_IF
		 IF bEnable = FALSE THEN iState := 0; END_IF
		 
	20 : //Wait handshake Stations
		 IF aStations[iStation].Sequence1(TRUE) THEN
			 aStations[iStation].Sequence1(FALSE);
			 iState := iState + 10;
		 END_IF
		 IF bEnable = FALSE THEN iState := 0; END_IF
		 	
	30 : //Go to Next Stations
		 iStation := iStation + 1;
		 IF aStations[iStation].stCfg.sName = '' THEN iStation := 1; END_IF
		 iState := SEL(bEnable, 0, 10);

 END_CASE
 Sequence1 := bBusy;
END_METHOD

END_FUNCTION_BLOCK

// ---- POUs/XTS/FB_Station.TcPOU
FUNCTION_BLOCK FB_Station
VAR_IN_OUT
	 //ax						: ARRAY [1..Tc3_XTS_Utility.TcIoXtsEnvironmentParameterList.MaxXtsMoversPerXpu] OF FB_Mover;	//Movers
END_VAR
VAR_INPUT
	stCfg 					: stStationCfg;
	udiNumMovers			: UDINT;		//Number of Movers into the system
	lrPartLength			: LREAL;
	bInvertPolarity			: BOOL;
END_VAR
VAR_OUTPUT
	udiNumMoversIn			: UDINT;		//Number of Movers into station
END_VAR
VAR
	
END_VAR
VAR CONSTANT
	START_POSITION_ON_PART_STATION 	: DWORD := 16#03080272;
	END_POSITION_ON_PART_STATION 	: DWORD := 16#03080273;
	STOP_POSITIONS_STATION 			: DWORD := 16#0308028D;
END_VAR

METHOD Sequence1 : BOOL
VAR_INPUT
	bExecute : BOOL;
END_VAR
VAR_OUTPUT
	bBusy	: BOOL;
	bError	: BOOL;
	bErrorID: BOOL;
END_VAR
VAR_INST
	iState 	: INT;
	m_bBusy	: BOOL;
	i		: UDINT;
	fbTON	: TON;
END_VAR
IF bExecute = FALSE THEN iState := 0; END_IF
CASE iState OF
	0 :
		IF bExecute THEN
			fbTON(IN := FALSE);
			iState := iState + 10;
		END_IF

	10 : //Check for movers between previous station position and start position
		 fbTON(IN := TRUE, PT := REAL_TO_TIME(stCfg.lrProcessingTime*1000.0));
		IF fbTON.Q THEN
			iState := iState + 10;
		END_IF
		
	20 : //Done
		Sequence1 := TRUE;
		IF bExecute = FALSE THEN
			iState := 0;
		END_IF
	
END_CASE
END_METHOD

METHOD SetStationInfo : BOOL
VAR_INPUT
	bExecute		: BOOL;
	OTCID			: DWORD;
END_VAR
VAR_INST
	iState 	 		: INT;
	fbADSWrite 		: adswrite;
	lrStartPos		: LREAL;
	lrEndPos		: LREAL;
	aStopPos		: ARRAY [1..3] OF LREAL;
	lrTmp			: LREAL;
	aTmp			: ARRAY [1..3] OF LREAL;
	lrDistance		: LREAL;
END_VAR

CASE iState OF
	0 : 
		IF bExecute THEN
			fbADSWrite(WRITE:= FALSE);
			iState 	:= iState + 1;
		END_IF
	
	1 : //Write Init position
		lrStartPos 	:= SEL(bInvertPolarity, stCfg.lrStartPosition, lrPartLength - stCfg.lrEndPosition);
		lrEndPos 	:= SEL(bInvertPolarity, stCfg.lrEndPosition, lrPartLength - stCfg.lrStartPosition);
		fbADSWrite(
			NETID:= , 
			PORT:= 350, 
			IDXGRP:= OTCID, 
			IDXOFFS:= START_POSITION_ON_PART_STATION, 
			LEN:= SIZEOF(lrStartPos), 
			SRCADDR:= ADR(lrStartPos), 
			WRITE:= TRUE, 
			TMOUT:= , 
			BUSY=> , 
			ERR=> , 
			ERRID=> );
	
		IF fbADSWrite.BUSY = FALSE AND fbADSWrite.ERR = FALSE THEN
			fbADSWrite(WRITE := FALSE);
			iState := iState + 1;
		END_IF	
			
	2 : //Write End Position
		fbADSWrite(
			NETID:= , 
			PORT:= 350, 
			IDXGRP:= OTCID, 
			IDXOFFS:= END_POSITION_ON_PART_STATION, 
			LEN:= SIZEOF(lrEndPos), 
			SRCADDR:= ADR(lrEndPos), 
			WRITE:= TRUE, 
			TMOUT:= , 
			BUSY=> , 
			ERR=> , 
			ERRID=> );
	
		IF fbADSWrite.BUSY = FALSE AND fbADSWrite.ERR = FALSE THEN
			fbADSWrite(WRITE := FALSE);
			iState := iState + 1;
		END_IF
		
	3 : //Write Stop Positions
		aStopPos[1] := SEL(bInvertPolarity, stCfg.lrStopPosition[1], (stCfg.lrEndPosition - stCfg.lrStartPosition) - stCfg.lrStopPosition[1]); 
		aStopPos[2] := SEL(bInvertPolarity, stCfg.lrStopPosition[2], (stCfg.lrEndPosition - stCfg.lrStartPosition) - stCfg.lrStopPosition[2]); 
		aStopPos[3] := SEL(bInvertPolarity, stCfg.lrStopPosition[3], (stCfg.lrEndPosition - stCfg.lrStartPosition) - stCfg.lrStopPosition[3]); 
		IF stCfg.uiNumStopPositions = 1 THEN
			aTmp[1] := aStopPos[1];
			aTmp[2] := aStopPos[1];
			aTmp[3] := aStopPos[1];
		ELSIF stCfg.uiNumStopPositions = 2 THEN
			aTmp[1] := SEL(bInvertPolarity, aStopPos[1], aStopPos[2]);
			aTmp[2] := SEL(bInvertPolarity, aStopPos[2], aStopPos[1]);
			aTmp[3] := SEL(bInvertPolarity, aStopPos[2], aStopPos[1]);
		ELSIF stCfg.uiNumStopPositions = 3 THEN
			aTmp[1] := SEL(bInvertPolarity, aStopPos[1], aStopPos[3]);
			aTmp[2] := SEL(bInvertPolarity, aStopPos[2], aStopPos[2]);
			aTmp[3] := SEL(bInvertPolarity, aStopPos[3], aStopPos[1]);
		ELSE
			aTmp[1]	:= 0.0;
			aTmp[2] := 0.0;
			aTmp[3] := 0.0;
		END_IF
		fbADSWrite(
			NETID:= , 
			PORT:= 350, 
			IDXGRP:= OTCID, 
			IDXOFFS:= STOP_POSITIONS_STATION, 
			LEN:= SIZEOF(aTmp), 
			SRCADDR:= ADR(aTmp), 
			WRITE:= TRUE, 
			TMOUT:= , 
			BUSY=> , 
			ERR=> , 
			ERRID=> );
	
		IF fbADSWrite.BUSY = FALSE AND fbADSWrite.ERR = FALSE THEN
			fbADSWrite(WRITE := FALSE);
			iState := iState + 1;
		END_IF
		
	4 : //Job Done
		SetStationInfo := TRUE;
		IF bExecute = FALSE THEN
			iState := 0;
		END_IF
	
END_CASE
END_METHOD

END_FUNCTION_BLOCK

// ---- POUs/XTS/MC_MoveAbsoluteTimeCA.TcPOU
FUNCTION_BLOCK MC_MoveAbsoluteTimeCA 
VAR_IN_OUT
	Axis					: AXIS_REF; 
END_VAR
VAR_INPUT
	bExecute				: BOOL;
	lrPosition 				: LREAL;
	lrTime 					: LREAL;
END_VAR
VAR_OUTPUT
	Done					: BOOL;		 
	Busy 					: BOOL;
	Active					: BOOL;
	CommandAborted 			: BOOL;
	Error					: BOOL;
	ErrorId					: UDINT;	
END_VAR
VAR
	iState					: INT;
	lrDistance				: LREAL;
	fbReadParamSet			: MC_ReadParameterSet := (Execute := TRUE);
	stParameter				: ST_AxisParameterSet;
	fbMoveAbsoluteCA		: MC_MoveAbsoluteCA;
END_VAR


CASE iState OF
	
	0 : IF bExecute THEN iState := iState + 1; END_IF
	
	1 :
		fbReadParamSet(Parameter := stParameter, Axis := Axis, Execute := TRUE);
		IF fbReadParamSet.Done THEN
			iState := iState + 1;
		END_IF
	2 :
		lrDistance := Tc2_Math.LMOD(lrPosition - axis.NcToPlc.ModuloSetPos + stParameter.fEncModuloFactor, stParameter.fEncModuloFactor);
		IF ABS(lrDistance) < 0.5 OR ABS(lrDistance-stParameter.fEncModuloFactor) < 0.5 THEN
			Done := TRUE;
			IF bExecute = FALSE THEN 
				fbMoveAbsoluteCA.Execute := FALSE;
				Done := FALSE;
				iState := 0; 
			END_IF
		ELSE 
			IF lrDistance < 0 THEN lrDistance := lrDistance + stParameter.fEncModuloFactor; END_IF
			fbMoveAbsoluteCA.Position		:= lrPosition;
			fbMoveAbsoluteCA.Velocity 		:= (lrDistance * 2.0) / lrTime;
			fbMoveAbsoluteCA.Acceleration 	:= (fbMoveAbsoluteCA.Velocity * 4.0) / lrTime;
			fbMoveAbsoluteCA.Deceleration 	:= (fbMoveAbsoluteCA.Velocity * 4.0) / lrTime;
			fbMoveAbsoluteCA.Jerk			:= (fbMoveAbsoluteCA.Acceleration * 4.0) / lrTime;
			fbMoveAbsoluteCA.Direction		:= tc3_mc3Definitions.MC_DIRECTION.mcDirectionPositive;
			iState := iState + 1;
		END_IF
		
	3 : //Execute
		fbMoveAbsoluteCA.Execute := TRUE;
		Done := fbMoveAbsoluteCA.Done;
		IF bExecute = FALSE THEN 
			fbMoveAbsoluteCA.Execute := FALSE;
			Done := FALSE;
			iState := 0; 
		END_IF
	
END_CASE

fbMoveAbsoluteCA(
	Axis:= Axis, 
	Execute:= , 
	ContinuousUpdate:= , 
	Position:= , 
	Velocity:= , 
	Acceleration:= , 
	Deceleration:= , 
	Jerk:= , 
	Gap:= , 
	BufferMode:= , 
	Direction:= , 
	Options:= , 
	Done=> , 
	Busy=> Busy, 
	Active=> Active, 
	CommandAborted=> CommandAborted, 
	Error=> Error, 
	ErrorId=> ErrorId);

END_FUNCTION_BLOCK

// ---- POUs/XTS/MC_JogCA.TcPOU
FUNCTION_BLOCK MC_JogCA EXTENDS MC_Jog
VAR_INPUT
END_VAR
VAR_OUTPUT
END_VAR
VAR
	fbMoveRelativeCA 	: MC_MoveRelativeCA;
	fbHaltCA 			: MC_HaltCA;
	fbReadParameterSet	: MC_ReadParameterSet;
	stParameters		: st_axisparameterset;
	Old_bJogForward		: BOOL;
	Old_bJogBackwards	: BOOL;
	nState				: (IDLE, STARTING, EXECUTE, STOPPING, RESETING, ABORTED);
	bBackwards			: BOOL;
END_VAR


CASE nState OF
	
	IDLE://
		IF JogForward AND Old_bJogForward = FALSE THEN nState := RESETING; bBackwards := FALSE; Busy := TRUE; END_IF
		IF JogBackwards AND Old_bJogBackwards = FALSE THEN nState := RESETING; bBackwards := TRUE; Busy := TRUE; END_IF
		IF JogForward = FALSE AND JogBackwards = FALSE THEN Done := FALSE; END_IF
		
	RESETING:
		fbReadParameterSet(Parameter := stParameters, Axis := Axis, Execute := FALSE); 
		fbMoveRelativeCA(Axis := Axis, Execute := FALSE);	
		fbHaltCA(Axis := Axis, Execute := FALSE);
		nState := STARTING;
		
	STARTING:
	
		CASE Mode OF
			E_JogMode.MC_JOGMODE_CONTINOUS:
				fbReadParameterSet(Parameter := stParameters, Axis := Axis, Execute := TRUE, Error => Error, ErrorID => ErrorID); 
				fbMoveRelativeCA.Distance  	:= SEL(bBackwards, stParameters.fEncModuloFactor, -stParameters.fEncModuloFactor);
				fbMoveRelativeCA.Velocity	:= Velocity;
				IF fbReadParameterSet.Done THEN
					nState := EXECUTE;
				END_IF
				IF Error THEN nState := ABORTED; END_IF
			E_JogMode.MC_JOGMODE_INCHING:
        		//
			E_JogMode.MC_JOGMODE_INCHING_MODULO:  
        		//
			E_JogMode.MC_JOGMODE_STANDARD_FAST: 
				fbReadParameterSet(Parameter := stParameters, Axis := Axis, Execute := TRUE, Error => Error, ErrorID => ErrorID); 
				fbMoveRelativeCA.Distance  	:= SEL(bBackwards, stParameters.fEncModuloFactor, -stParameters.fEncModuloFactor);
				fbMoveRelativeCA.Velocity	:= stParameters.fVeloFastManual;
				IF fbReadParameterSet.Done THEN
					nState := EXECUTE;
				END_IF
				IF Error THEN nState := ABORTED; END_IF
			E_JogMode.MC_JOGMODE_STANDARD_SLOW:
				fbReadParameterSet(Parameter := stParameters, Axis := Axis, Execute := TRUE, Error => Error, ErrorID => ErrorID); 
				fbMoveRelativeCA.Distance  	:= SEL(bBackwards, stParameters.fEncModuloFactor, -stParameters.fEncModuloFactor);
				fbMoveRelativeCA.Velocity	:= stParameters.fVeloSlowManual;
				IF fbReadParameterSet.Done THEN
					nState := EXECUTE;
				END_IF
				IF Error THEN nState := ABORTED; END_IF
		END_CASE
		
	EXECUTE:

		fbMoveRelativeCA(Axis := Axis, Execute := TRUE, Active => Active, Error => Error, ErrorID => ErrorID, CommandAborted => CommandAborted, Done => Done);	
		IF (JogForward = FALSE AND bBackwards = FALSE) OR (JogBackwards = FALSE AND bBackwards = TRUE) THEN
			nState := STOPPING;
		END_IF
		IF Error THEN nState := ABORTED; END_IF
	
	STOPPING:
	
		fbHaltCA(Axis := Axis, Execute := TRUE, Error => Error, ErrorID => ErrorID, CommandAborted => CommandAborted, Done => Done);
		IF Error THEN nState := ABORTED; END_IF
		IF Done THEN nState := IDLE; Busy := FALSE; END_IF
		
	ABORTED:
		Active 	:= FALSE;
		Busy 	:= FALSE;
		Done	:= FALSE;
		IF (JogForward = FALSE AND bBackwards = FALSE) OR (JogBackwards = FALSE AND bBackwards = TRUE) THEN
			Error 	:= FALSE;
			nState 	:= IDLE;
		END_IF
	
END_CASE

Old_bJogForward := JogForward;

END_FUNCTION_BLOCK

// ---- POUs/XTS/FB_GroupCA.TcPOU
FUNCTION_BLOCK FB_GroupCA
VAR_IN_OUT
	ax					: ARRAY [1..Tc3_XTS_Utility.TcIoXtsEnvironmentParameterList.MaxXtsMoversPerXpu] OF fb_Mover;
END_VAR
VAR_INPUT
	fbXPUGroupCA		: FB_Mc2CaGroup;
END_VAR
VAR_OUTPUT
	eGroupState			: MC_GROUP_STATE;
	bAllStandStill		: BOOL;
	bError				: BOOL;
END_VAR
VAR 
	//Function Blocks
	ag					: AXES_GROUP_REF;
	fbEnable			: MC_GroupEnable;
	fbDisable			: MC_GroupDisable;
	fbHalt				: MC_GroupHalt;
	fbUnGroupAll		: MC_UngroupAllAxes;
	fbGroupStop			: MC_GroupStop;
	fbReset				: MC_GroupReset;
	fbState				: MC_GroupReadStatus;
END_VAR

fbEnable(
	AxesGroup:= ag, 
	Execute:= , 
	Done=> , 
	Busy=> , 
	Error=> , 
	ErrorId=> );
	
fbDisable(
	AxesGroup:= ag, 
	Execute:= , 
	Done=> , 
	Busy=> , 
	Error=> , 
	ErrorId=> );
	
fbGroupStop(
	AxesGroup:= ag, 
	Execute:= , 
	Deceleration:= , 
	Jerk:= , 
	Done=> , 
	Busy=> , 
	Active=> , 
	CommandAborted=> , 
	Error=> , 
	ErrorId=> );
	
fbHalt(
	AxesGroup:= ag, 
	Execute:= , 
	Deceleration:= , 
	Jerk:= , 
	Done=> , 
	Busy=> , 
	Active=> , 
	CommandAborted=> , 
	Error=> , 
	ErrorId=> );
	
fbUnGroupAll(
	AxesGroup:= ag, 
	Execute:= , 
	Done=> , 
	Busy=> , 
	Error=> , 
	ErrorId=> );
	
fbReset(
	AxesGroup:= ag, 
	Execute:= , 
	Done=> , 
	Busy=> , 
	Error=> , 
	ErrorId=> );
	
fbState(
	AxesGroup:= ag, 
	Enable:= TRUE, 
	Valid=> , 
	Busy=> , 
	GroupMoving=> , 
	GroupHoming=> , 
	GroupErrorStop=> , 
	GroupNotReady=> , 
	GroupStandby=> , 
	GroupStopping=> , 
	GroupDisabled=> , 
	AllAxesStanding=> , 
	ConstantVelocity=> , 
	Accelerating=> , 
	Decelerating=> , 
	InPosition=> , 
	Error=> , 
	ErrorId=> );
	
IF fbState.GroupDisabled THEN
	eGroupState := MC_GROUP_STATE.mcGroupStateDisabled;
ELSIF fbState.GroupErrorStop THEN
	eGroupState := MC_GROUP_STATE.mcGroupStateErrorStop;
ELSIF fbState.GroupHoming THEN
	eGroupState := MC_GROUP_STATE.mcGroupStateHoming;
ELSIF fbState.GroupMoving THEN
	eGroupState := MC_GROUP_STATE.mcGroupStateMoving;
ELSIF fbState.GroupNotReady THEN
	eGroupState := MC_GROUP_STATE.mcGroupStateNotReady;
ELSIF fbState.GroupStandby THEN
	eGroupState := MC_GROUP_STATE.mcGroupStateStandby;
ELSIF fbState.GroupStopping THEN
	eGroupState := MC_GROUP_STATE.mcGroupStateStopping;
ELSIF fbState.GroupStandby THEN
	eGroupState := MC_GROUP_STATE.mcGroupStateSuspended;
ELSE
	eGroupState := MC_GROUP_STATE.mcGroupStateInvalid;
END_IF
bError := eGroupState = mc_group_state.mcGroupStateErrorStop;
bAllStandStill := fbState.AllAxesStanding;

METHOD m_clearCmd : BOOL
VAR_INPUT
END_VAR
m_halt(FALSE);
m_reset(FALSE);
m_ungroupall(FALSE);
m_enable(FALSE);
m_disable(FALSE);
END_METHOD

METHOD m_disable : bool
VAR_INPUT
	bExecute : BOOL;
END_VAR
fbDisable.Execute 	:= bExecute;
m_disable			:= fbDisable.Done;
END_METHOD

METHOD m_enable : bool
VAR_INPUT
	bEnable : BOOL;
END_VAR
fbEnable.Execute 	:= bEnable;
m_enable			:= fbEnable.Done;
END_METHOD

METHOD m_halt : bool
VAR_INPUT
	bExecute : BOOL;
END_VAR
fbHalt.Execute 		:= bExecute;
m_halt				:= fbHalt.Done;
END_METHOD

METHOD m_reset : bool
VAR_INPUT
	bREset : BOOL;
END_VAR
fbReset.Execute := bREset;
m_reset			:= fbReset.Done;
END_METHOD

METHOD m_ungroupall : bool
VAR_INPUT
	bExecute :BOOL;
END_VAR
fbUnGroupAll.Execute 	:= bExecute;
m_ungroupall			:= fbUnGroupAll.Done;
END_METHOD

END_FUNCTION_BLOCK

// ---- GlobalTextList.TcGTLO
TEXTLIST GlobalTextList
  73 = '%5.2f'
  340 = '%d'
  772 = 'AllStandStill'
  210 = 'AUTO'
  154 = 'AUTOMATIC'
  2693 = 'Automatic'
  142 = 'CONTROL'
  992 = 'ENABLE'
  267 = 'End Position'
  605 = 'Error'
  2378 = 'Init Done'
  146 = 'JOG +'
  2714 = 'JOG -'
  124 = 'Log: %s'
  1878 = 'MANUAL'
  2735 = 'Manual'
  2444 = 'MOVE'
  1070 = 'Mover Selection'
  265 = 'Name'
  270 = 'Num Stop Positions'
  958 = 'Number of Stations'
  269 = 'Processing Time'
  176 = 'RESET'
  266 = 'Start Position'
  1046 = 'Station Selection'
  570 = 'STATUS'
  268 = 'Stop Position'
  3040 = 'Stop Position Selection'
  448 = 'Target Position'
  809 = 'Target Velocity'
  3087 = 'TEACH STATION'
  271 = 'Travel Time'
END_TEXTLIST

// ---- VISUs/GlobalTextList_1.TcGTLO
TEXTLIST GlobalTextList_1
  81 = ''
  752 = '%'
  221 = '%3.3f'
  249 = '%3.3f [s]'
  73 = '%5.2f'
  853 = '%5.3f'
  1155 = '%5.3f ms'
  340 = '%d'
  844 = '%f2.3'
  967 = '%f5.2'
  16 = '%s'
  1814 = '%S'
  688 = '%x'
  760 = '-'
  1799 = '----'
  1817 = '-----'
  363 = '1'
  67 = '10'
  1584 = '11'
  1164 = '12'
  184 = '13'
  1855 = '14'
  603 = '15'
  144 = '2'
  761 = '3'
  538 = '4'
  264 = '5'
  1091 = '6'
  1096 = '7'
  1571 = '8'
  1397 = '9'
  277 = 'ACC'
  587 = 'Acceleration'
  152 = 'Acceleration: %5.2f uu'
  233 = 'Acceleration: %5.2f uu/s2'
  346 = 'ACK'
  2022 = 'Ack'
  401 = 'Ack Mode'
  1577 = 'Acknowlage'
  397 = 'Act Pos: %5.2f uu'
  612 = 'ActAcc: %5.2f uu'
  248 = 'ActAcc: %5.2f uu/s2'
  742 = 'ActPos'
  696 = 'ActPos: %5.2f uu'
  1837 = 'Actual Mode'
  1778 = 'Actual Mode: %s'
  504 = 'ActVelo'
  704 = 'ActVelo: %5.2f uu'
  400 = 'ActVelo: %5.2f uu/s'
  691 = 'ADD'
  288 = 'ADD TO GROUP'
  713 = 'ALL'
  606 = 'APPLY'
  1404 = 'APPLY CFG'
  147 = 'aStations[2]'
  187 = 'aStations[3]'
  210 = 'AUTO'
  154 = 'AUTOMATIC'
  2693 = 'Automatic'
  717 = 'Axis ID: %d'
  485 = 'axis running'
  300 = 'bBestFit'
  456 = 'Best Fit'
  108 = 'BEST FIT'
  112 = 'BestFit'
  341 = 'Buffer:'
  237 = 'BUILD'
  459 = 'Busy'
  20 = 'Cancel'
  1815 = 'CANCEL'
  585 = 'Command'
  1081 = 'Command: %s'
  124 = 'COMPLETE'
  1574 = 'CONFIG'
  360 = 'CONFIGURATION'
  1010 = 'Configuration'
  139 = 'Control'
  142 = 'CONTROL'
  1867 = 'CREATE'
  278 = 'CTRL'
  988 = 'DC link '
  2064 = 'Deceleration: %5.2f uu'
  856 = 'Deceleration: %5.2f uu/s2'
  366 = 'DEFAULT'
  367 = 'Default Gap'
  1980 = 'DELETE'
  928 = 'Destination Station'
  1457 = 'DIAG'
  1716 = 'Direction'
  2867 = 'Direction:'
  885 = 'DISABLE'
  762 = 'Disable'
  869 = 'Done'
  37 = 'E'
  992 = 'ENABLE'
  737 = 'ENABLE C'
  750 = 'Enable Control'
  1492 = 'ENABLE CONTROL'
  1711 = 'ENABLE FORWARD'
  2101 = 'ENABLE NEGATIVE'
  296 = 'ENABLE POSITIVE'
  1013 = 'ENABLE REVERSE'
  58 = 'Enable Visu Control'
  905 = 'ENC'
  1459 = 'END'
  222 = 'END POS'
  386 = 'End Position'
  605 = 'Error'
  1623 = 'Error ID'
  2237 = 'Error ID: %i'
  2498 = 'Error ID: %x'
  1092 = 'ErrorID'
  661 = 'ErrorID %x'
  2074 = 'ErrorID: %5.2f'
  1737 = 'ErrorID: %x'
  930 = 'EXECUTE'
  1004 = 'Execute'
  1054 = 'Extra Cfg.'
  797 = 'F1 --'
  751 = 'F2 -'
  932 = 'F3 +'
  447 = 'F4 ++'
  241 = 'F4++'
  377 = 'F5'
  151 = 'F6'
  301 = 'F8'
  1345 = 'FILE'
  842 = 'From Station'
  345 = 'Functions'
  622 = 'Gap'
  265 = 'Gap: %5.2f uu'
  148 = 'GENERAL'
  1248 = 'GROUP'
  39 = 'GROUP ALL'
  78 = 'GROUP CA'
  1332 = 'Group CA'
  123 = 'GROUP STATE:'
  767 = 'Group State: %s'
  787 = 'GroupCA'
  166 = 'HALT'
  1759 = 'HALT CA'
  719 = 'HandShake Offset'
  714 = 'HandShakeOffset'
  53 = 'Home'
  1348 = 'HOME'
  1416 = 'ID'
  2378 = 'Init Done'
  777 = 'Jerk'
  630 = 'JERK'
  1973 = 'JOG'
  146 = 'JOG +'
  2714 = 'JOG -'
  2062 = 'JOG CA'
  133 = 'Jog Mode'
  2110 = 'Join GapGap'
  858 = 'LOAD'
  1730 = 'LOCAL INTERLOCK'
  196 = 'loooooooool'
  1878 = 'MANUAL'
  2735 = 'Manual'
  1218 = 'Mask Control'
  138 = 'Members'
  134 = 'Message: %s'
  887 = 'Mode'
  574 = 'MODES'
  883 = 'Modo Operación'
  0 = 'Module'
  60 = 'MODULES'
  2444 = 'MOVE'
  2277 = 'MOVE ABSOLUTE'
  369 = 'MOVE ABSOLUTE CA'
  234 = 'MOVE ALL'
  1546 = 'MOVE ONE'
  783 = 'MOVE ONE FW'
  1344 = 'MOVE RELATIVE CA'
  186 = 'Move Time'
  1000 = 'MOVE TIME'
  55 = 'Mover'
  1117 = 'Mover ID: %s'
  455 = 'Mover In Station'
  1070 = 'Mover Selection'
  217 = 'Mover Selection Control'
  329 = 'MOVER STATE:'
  728 = 'MOVERS'
  972 = 'Movers Join Gap'
  1363 = 'Movers Waiting'
  966 = 'NAME'
  178 = 'Name'
  645 = 'NAMES'
  299 = 'NEGATIVE'
  996 = 'Negative Limit: %5.2f uu'
  192 = 'Negative Software Limit'
  347 = 'NEW'
  165 = 'No'
  271 = 'Num Active'
  24 = 'Num Stop Positions'
  267 = 'Num Stops'
  908 = 'NumActive'
  958 = 'Number of Stations'
  632 = 'Number of stations: %d'
  766 = 'Ok'
  149 = 'OK'
  492 = 'ONLINE'
  1859 = 'OPEN FROM'
  596 = 'Operation Mode'
  472 = 'Origin Station'
  893 = 'Overall current'
  684 = 'Part'
  2092 = 'PARTS'
  862 = 'PAUSE'
  843 = 'POS'
  907 = 'Posiciones de Parada'
  954 = 'Posición 1'
  439 = 'Posición 2'
  712 = 'Posición 3'
  794 = 'Posición Parada'
  870 = 'Position'
  2475 = 'Position: %5.2f'
  726 = 'Position: %5.2f uu'
  1406 = 'POSITIVE'
  402 = 'Positive Limit: %5.2f uu'
  137 = 'Positive Software Limit'
  812 = 'POWER'
  314 = 'POWER ALL'
  1269 = 'PROCESS'
  582 = 'Process Time'
  473 = 'Processing Time'
  581 = 'ProcessTime'
  754 = 'PRODUCTION'
  394 = 'R'
  1418 = 'READ'
  541 = 'RECIPE'
  294 = 'Recipe Name'
  997 = 'RECIPES'
  200 = 'Request Mode'
  935 = 'RESEE'
  176 = 'RESET'
  216 = 'Reset axis'
  145 = 'RESTART'
  4 = 'Routes'
  949 = 'ROUTES'
  702 = 'Running'
  819 = 'SAVE'
  76 = 'SAVE AS'
  395 = 'SET'
  310 = 'Set Acc'
  92 = 'Set Jerk'
  888 = 'Set Pos: %5.2f uu'
  1573 = 'Set Position: %5.2f uu'
  963 = 'Set Velo'
  2851 = 'Set Velocity: %5.2f uu'
  15 = 'SetAcc'
  140 = 'SetAcc: %5.2f uu/s2'
  646 = 'Some error into axis'
  1234 = 'START'
  749 = 'START POS'
  51 = 'Start Position'
  1158 = 'STATE'
  1305 = 'State'
  1425 = 'State: %s'
  392 = 'Station'
  1046 = 'Station Selection'
  1831 = 'STATION: %s'
  664 = 'Stations'
  141 = 'STATIONS'
  2091 = 'Status'
  286 = 'STOP'
  692 = 'Stop Pos. 1'
  375 = 'Stop Pos. 2'
  465 = 'Stop Pos. 3'
  1729 = 'Stop Position'
  362 = 'Stop Position 1'
  357 = 'Stop Position 2'
  1064 = 'Stop Position 3'
  3040 = 'Stop Position Selection'
  238 = 'Stop Positions'
  1469 = 'Suspend'
  792 = 'Target Acc: %5.2f uu'
  868 = 'Target Pos: %5.2f uu'
  448 = 'Target Position'
  757 = 'Target Time: %5.2f uu'
  720 = 'Target Velo: %5.2f uu'
  809 = 'Target Velocity'
  3087 = 'TEACH STATION'
  592 = 'TEACHING'
  199 = 'To Station'
  1396 = 'Total Axis'
  599 = 'Total Axis: %d'
  919 = 'Track'
  674 = 'Travel Time'
  1443 = 'UN PAUSE'
  1569 = 'UNBUILD'
  1900 = 'UPDATE DIAG'
  3005 = 'UTILITIES'
  1235 = 'UTILITY'
  964 = 'VALUES'
  1059 = 'VELO'
  878 = 'Velocity'
  2644 = 'Velocity %5.2f uu'
  2099 = 'Velocity: %5.2f uu'
  153 = 'Velocity: %5.2f uu/s'
  625 = 'VIEWER'
  57 = 'VISU MODE'
  623 = 'Waiting Time'
  150 = 'WIZARD'
  1408 = 'WRITE'
  520 = 'X'
  851 = 'XPU'
  1038 = 'Xpu'
  848 = 'XTS'
  855 = 'XTS Processing Unit - Control'
  1918 = 'XTS Processing Unit - Group CA'
  753 = 'XTS Processing Unit - Movers'
  1176 = 'XTS Processing Unit - Stations'
  3469 = 'XTS Utility'
  344 = 'XTS VIEWER'
  1135 = 'xts.aStations[7]'
  1005 = 'Yes'
END_TEXTLIST

// ---- VISUs/GlobalTextList_2.TcGTLO
TEXTLIST GlobalTextList_2
  73 = '%5.2f'
  340 = '%d'
  772 = 'AllStandStill'
  210 = 'AUTO'
  154 = 'AUTOMATIC'
  2693 = 'Automatic'
  142 = 'CONTROL'
  992 = 'ENABLE'
  863 = 'End Position'
  605 = 'Error'
  2378 = 'Init Done'
  146 = 'JOG +'
  2714 = 'JOG -'
  832 = 'Log: %5s'
  124 = 'Log: %s'
  1878 = 'MANUAL'
  2735 = 'Manual'
  2444 = 'MOVE'
  1070 = 'Mover Selection'
  861 = 'Name'
  866 = 'Num Stop Positions'
  958 = 'Number of Stations'
  865 = 'Processing Time'
  176 = 'RESET'
  862 = 'Start Position'
  1046 = 'Station Selection'
  570 = 'STATUS'
  864 = 'Stop Position'
  3040 = 'Stop Position Selection'
  448 = 'Target Position'
  809 = 'Target Velocity'
  3087 = 'TEACH STATION'
  867 = 'Travel Time'
END_TEXTLIST

// ---- VISUs/TextList/AxisState_txt.TcTLO
TEXTLIST AxisState_txt
  0 = 'INVALID'
  1 = 'DISABLED'
  2 = 'STANDSTILL'
  3 = 'ERROR STOP'
  4 = 'STOPPING'
  5 = 'HOMING'
  6 = 'DISCRETE MOTION'
  7 = 'CONTINIOUS MOTION'
  8 = 'SYNCHRONIZED MOTION'
   = ''
END_TEXTLIST

// ---- VISUs/TextList/GroupState_txt.TcTLO
TEXTLIST GroupState_txt
  0 = 'INVALID'
  1 = 'DISABLED'
  2 = 'STANDBY'
  3 = 'MOVING'
  4 = 'STOPPING'
  5 = 'ERROR STOP'
  6 = 'HOMING'
  7 = 'NOT READY'
  8 = 'SUSPENDED'
   = ''
END_TEXTLIST

// ---- VISUs/TextList/MoversMode_txt.TcTLO
TEXTLIST MoversMode_txt
  1 = 'Single'
  2 = 'Double'
  3 = 'Triple'
   = ''
END_TEXTLIST

// ---- VISUs/TextList/PML_Modes_txt.TcTLO
TEXTLIST PML_Modes_txt
  0 = 'Undefined'
  1 = 'Production'
  2 = 'Manual'
   = ''
END_TEXTLIST

// ---- VISUs/TextList/StationAckMode_txt.TcTLO
TEXTLIST StationAckMode_txt
  0 = 'Time'
  1 = 'External Ack'
   = ''
END_TEXTLIST

// ---- VISUs/Visualization.TcVIS
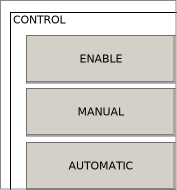
VISUALIZATION Visualization  // 177x190
    Frame (0,0 177x190)
        shows XTS_System_VISU(xts := MAIN.fbXTSSystem)
END_VISUALIZATION

// ---- VISUs/XTS_System_VISU.TcVIS
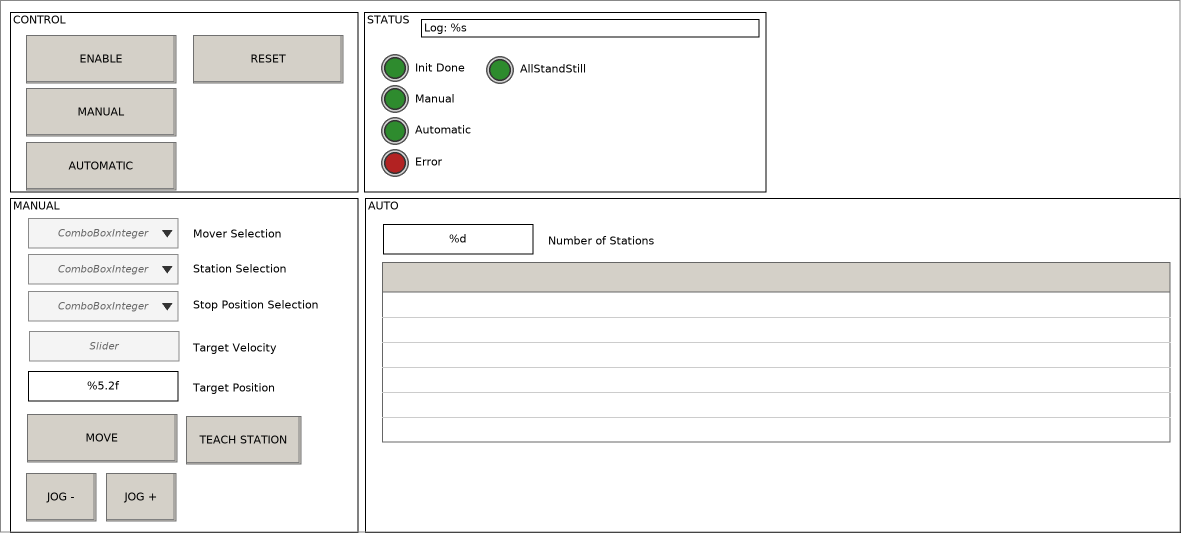
VISUALIZATION XTS_System_VISU  // 1181x533
VAR_IN_OUT
	xts : XTS_System;
END_VAR
    Rectangle (364,12 402x180), "STATUS"
    Rectangle (10,12 348x180), "CONTROL"
    Rectangle (10,198 348x335), "MANUAL"
    Button (26,35 150x48), "ENABLE"
        toggle xts.bEnable
    Button (26,88 150x48), "MANUAL"
        toggle xts.bManual
    Button (26,142 150x48), "AUTOMATIC"
        toggle xts.bAutomatic
    Lamp1 (379,52 32x32), variable: xts.bInitDone, style: Lamp-Lamp1-Green
    Label (412,53 110x30), "Init Done"
    ComboBoxInteger (28,218 150x30), variable: xts.udiMoverSelection
    ComboBoxInteger (28,254 150x30), variable: xts.udiStationSelection
    Label (190,219 150x30), "Mover Selection"
    Label (190,254 150x30), "Station Selection"
    ComboBoxInteger (28,291 150x30), variable: xts.udiStopPositionSelection
    Label (190,290 150x30), "Stop Position Selection"
    Button (27,414 150x48), "MOVE"
        tap xts.bManualMove
    Button (26,473 70x48), "JOG -"
        tap xts.bJogBackwards
    Button (106,473 70x48), "JOG +"
        tap xts.bJogForward
    Lamp1 (379,83 32x32), variable: xts.bInManual, style: Lamp-Lamp1-Green
    Label (412,84 110x30), "Manual"
    Lamp1 (379,115 32x32), variable: xts.bInAutomatic, style: Lamp-Lamp1-Green
    Label (412,115 110x30), "Automatic"
    Slider (29,331 150x30), variable: xts.lrTargetVelocity, scale 1..4000
    Label (190,333 150x30), "Target Velocity"
    Rectangle (28,371 150x30), "%5.2f", text variable: xts.lrTargetPosition
        OnMouseClick: write the text variable via Default
    Label (190,373 150x30), "Target Position"
    Button (186,416 115x48), "TEACH STATION"
        tap xts.bTeachStation
    Lamp1 (379,147 32x32), variable: xts.bError, style: Lamp-Lamp1-Red
    Label (412,147 110x30), "Error"
    Button (193,35 150x48), "RESET"
        tap xts.bReset
    Rectangle (365,198 816x335), "AUTO"
    Rectangle (383,224 150x30), "%d", text variable: xts.stCfg.udiNumStations
        OnMouseClick: write the text variable via Default
    Label (545,226 150x30), "Number of Stations"
    Table (382,262 788x180), data array: xts.stVisuStationsCfg
        p3854506369: xts.stVisuStationsCfg[INDEX].sName
        p1892666644: xts.stVisuStationsCfg[INDEX].lrStartPosition
        p338671338: xts.stVisuStationsCfg[INDEX].lrEndPosition
        p2170511999: xts.stVisuStationsCfg[INDEX].lrStopPosition
        p3723444502: xts.stVisuStationsCfg[INDEX].lrProcessingTime
        p1218418051: xts.stVisuStationsCfg[INDEX].uiNumStopPositions
        p746581629: xts.stVisuStationsCfg[INDEX].lrTravelTime
        p511219082: Start Position
        p1755163831: End Position
        p4092479075: Stop Position
        p2237128397: Processing Time
        p505689113: Num Stop Positions
        p1757482276: Travel Time
    Rectangle (421,19 338x18), "Log: %s", text variable: xts.sLog
        OnMouseClick: write the text variable via Default
    Lamp1 (484,54 32x32), variable: xts.bAllMoversStandStill, style: Lamp-Lamp1-Green
    Label (517,54 110x30), "AllStandStill"
END_VISUALIZATION
